FUNCTION_BLOCK VVI_VRP
  (* Standard: 61499-2 *)
  (* Version 0.1, 2014-00-19, Administrator, NE734EFZE6G0NVX *)
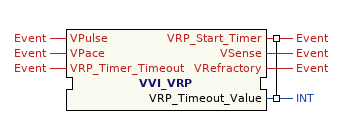
  EVENT_INPUT
    VPulse;
    VPace;
    VRP_Timer_Timeout;
  END_EVENT
  EVENT_OUTPUT
    VRP_Start_Timer WITH VRP_Timeout_Value;
    VSense;
    VRefractory;
  END_EVENT
  VAR_OUTPUT
    VRP_Timeout_Value : INT;
  END_VAR
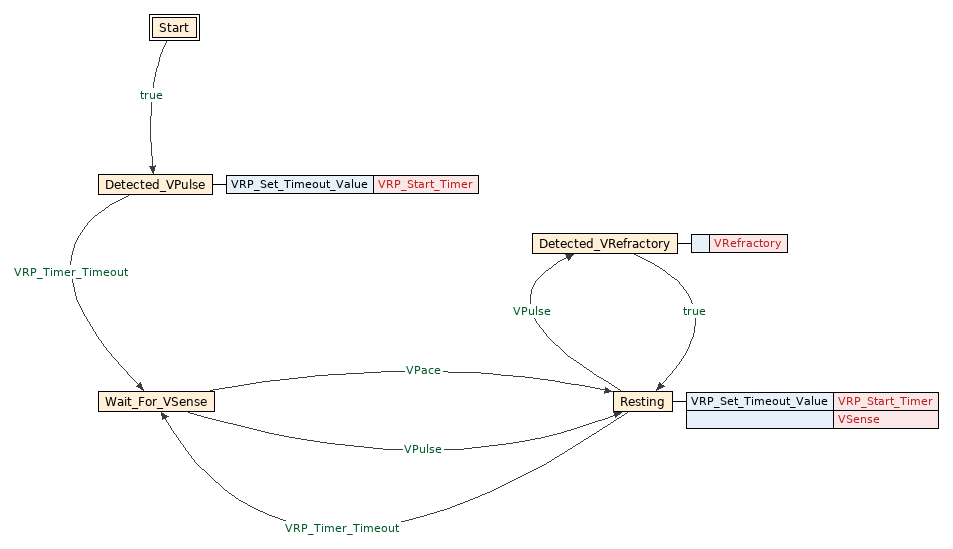
  EC_STATES
    Start;
    Wait_For_VSense;
    Resting : VRP_Set_Timeout_Value -> VRP_Start_Timer, -> VSense;
    Detected_VPulse : VRP_Set_Timeout_Value -> VRP_Start_Timer;
    Detected_VRefractory : -> VRefractory;
  END_STATES
  EC_TRANSITIONS
    Wait_For_VSense TO Resting := VPulse;
    Wait_For_VSense TO Resting := VPace;
    Resting TO Detected_VRefractory := VPulse;
    Resting TO Wait_For_VSense := VRP_Timer_Timeout;
    Start TO Detected_VPulse := true;
    Detected_VPulse TO Wait_For_VSense := VRP_Timer_Timeout;
    Detected_VRefractory TO Resting := true;
  END_TRANSITIONS
  ALGORITHM VRP_Set_Timeout_Value IN ST:
VRP_Timeout_Value := 300;
  END_ALGORITHM
END_FUNCTION_BLOCK
